Staubli VAL3: Staubli.pjx

--- Staubli.pjx ---
Parameters version=s7.9.1 stackSize=5000 millimeterUnit=true
Program file=decodeVelCfg.pgx
Program file=decodeVelCmd.pgx
Program file=decSetDrvPwrMsg.pgx
Program file=decWriSingIOMsg.pgx
Program file=encodeVelCfgAck.pgx
Program file=encodeVelCmdAck.pgx
Program file=encSetDrvPwrAck.pgx
Program file=encWriSingIOAck.pgx
Program file=init.pgx
Program file=initStaubliMsgs.pgx
Program file=start.pgx
Program file=stop.pgx
Data file=Staubli.dtx
Library alias=SimpleMsg path=Disk://ros_libs/SimpleMessage/SimpleMessage.pjx
Type name=_MotionMode path=./_MotionMode/MotionMode.pjx
Type name=_MsgTypeStaubli path=./_MsgTypeStaubli/MsgTypeStaubli.pjx
Type name=_VelocityType path=./_VelocityType/VelocityType.pjx
Type name=VelocityCmdMsg path=./VelocityCmdMsg/VelocityCmdMsg.pjx
Type name=VelocityCfgMsg path=./VelocityCfgMsg/VelocityCfgMsg.pjx
Type name=SetDrivePwrMsg path=./SetDrivePwrMsg/SetDrivePwrMsg.pjx
Type name=WriteSingIOMsg path=./WriteSingIOMsg/WriteSingIOMsg.pjx

--- Staubli.dtx ---
public SetDrivePwrMsg setDrvPwrAck
  [0]
    bool bDrivePower
    Body body
      [0]
        num nData
    Header header
      [0]
        num nCommType
        num nData[12]
        num nMsgType
        num nReplyCode
    Prefix prefix
      [0]
        num nData[4]
        num nLength
public SetDrivePwrMsg setDrvPwrMsg
  [0]
    bool bDrivePower
    Body body
      [0]
        num nData
    Header header
      [0]
        num nCommType
        num nData[12]
        num nMsgType
        num nReplyCode
    Prefix prefix
      [0]
        num nData[4]
        num nLength
public VelocityCfgMsg velCfgAck
  [0]
    Body body
      [0]
        num nData[68]
    Header header
      [0]
        num nCommType
        num nData[12]
        num nMsgType
        num nReplyCode
    Prefix prefix
      [0]
        num nData[4]
        num nLength = 76
    VelocityCfg velCfg
      [0]
        num nAccel
        num nCmdType
        num nRefFrameVec[6]
        num nRotVel
        num nToolVec[6]
        num nTransVel
public VelocityCfgMsg velCfgMsg
  [0]
    Body body
      [0]
        num nData[68]
    Header header
      [0]
        num nCommType
        num nData[12]
        num nMsgType
        num nReplyCode
    Prefix prefix
      [0]
        num nData[4]
        num nLength
    VelocityCfg velCfg
      [0]
        num nAccel
        num nCmdType
        num nRefFrameVec[6]
        num nRotVel
        num nToolVec[6]
        num nTransVel
public VelocityCmdMsg velCmdAck
  [0]
    Body body
      [0]
        num nData[32]
    Header header
      [0]
        num nCommType
        num nData[12]
        num nMsgType
        num nReplyCode
    Prefix prefix
      [0]
        num nData[4]
        num nLength = 44
    VelocityCmd velCmd
      [0]
        num nCmdType
        num nSeq
        num nVelVec[6]
public VelocityCmdMsg velCmdMsg
  [0]
    Body body
      [0]
        num nData[32]
    Header header
      [0]
        num nCommType
        num nData[12]
        num nMsgType
        num nReplyCode
    Prefix prefix
      [0]
        num nData[4]
        num nLength
    VelocityCmd velCmd
      [0]
        num nCmdType
        num nSeq
        num nVelVec[6]
public WriteSingIOMsg writeSingIOMsg
  [0]
    Body body
      [0]
        num nData[9]
    Header header
      [0]
        num nCommType
        num nData[12]
        num nMsgType
        num nReplyCode
    Prefix prefix
      [0]
        num nData[4]
        num nLength
    WriteSingleIO writeSingleIO
      [0]
        bool bState
        num nModuleId
        num nPin
public WriteSingIOMsg writeSingIOAck
  [0]
    Body body
      [0]
        num nData[9]
    Header header
      [0]
        num nCommType
        num nData[12]
        num nMsgType
        num nReplyCode
    Prefix prefix
      [0]
        num nData[4]
        num nLength
    WriteSingleIO writeSingleIO
      [0]
        bool bState
        num nModuleId
        num nPin
public _MotionMode MotionMode
  [0]
    num INVALID
    num JOINT_TRAJ = 1
    num VELOCITY_CTRL = 4
public _MsgTypeStaubli MsgType
  [0]
    num SET_DRIVE_POWER
    num VELOCITY_CFG = 1640
    num VELOCITY_CMD = 1641
    num READ_IO
    num WRITE_SINGLE_IO
public _VelocityType VelocityType
  [0]
    num INVALID
    num JOINT = 1
    num BASE_FRAME = 2
    num TOOL_FRAME = 3

--- decodeVelCfg.pgx ---
public program decodeVelCfg(bool& x_bFlag (dimensions=1))
  local num l_nIndex
  local num l_nRetVal
begin
  // Copyright (c) 2021, Institute for Factory Automation and Production Systems (FAPS)
  //
  // Licensed under the Apache License, Version 2.0 (the "License");
  // you may not use this file except in compliance with the License.
  // You may obtain a copy of the License at
  //
  //     http://www.apache.org/licenses/LICENSE-2.0
  //
  // Unless required by applicable law or agreed to in writing, software
  // distributed under the License is distributed on an "AS IS" BASIS,
  // WITHOUT WARRANTIES OR CONDITIONS OF ANY KIND, either express or implied.
  // See the License for the specific language governing permissions and
  // limitations under the License.


  // decode velocity configuration message body (data)

  // assume failure to decode
  velCfgAck.header.nReplyCode=SimpleMsg:ReplyCode.FAILURE


  // command type (frame or joint), 4 bytes
  l_nRetVal=fromBinary(velCfgMsg.body.nData,4,"-4l",velCfgMsg.velCfg.nCmdType)
  if (l_nRetVal!=1)
    x_bFlag=false
    return
  endIf

  // reference frame vector [6], 24 bytes
  for l_nIndex=0 to 5 step 1
    l_nRetVal=fromBinary(velCfgMsg.body.nData[(l_nIndex*4)+4],4,"4.0l",velCfgMsg.velCfg.nRefFrameVec[l_nIndex])
    if (l_nRetVal!=1)
      x_bFlag=false
      return
    endIf
  endFor

  // target tool vector [6], 24 bytes
  for l_nIndex=0 to 5 step 1
    l_nRetVal=fromBinary(velCfgMsg.body.nData[(l_nIndex*4)+28],4,"4.0l",velCfgMsg.velCfg.nToolVec[l_nIndex])
    if (l_nRetVal!=1)
      x_bFlag=false
      return
    endIf
  endFor

  // acceleration, 4 bytes
  l_nRetVal=fromBinary(velCfgMsg.body.nData[52],4,"4.0l",velCfgMsg.velCfg.nAccel)
  if (l_nRetVal!=1)
    x_bFlag=false
    return
  endIf

  // velocity, 4 bytes
  l_nRetVal=fromBinary(velCfgMsg.body.nData[56],4,"4.0l",velCfgMsg.velCfg.nVel)
  if (l_nRetVal!=1)
    x_bFlag=false
    return
  endIf

  // translational velocity, 4 bytes
  l_nRetVal=fromBinary(velCfgMsg.body.nData[60],4,"4.0l",velCfgMsg.velCfg.nTransVel)
  if (l_nRetVal!=1)
    x_bFlag=false
    return
  endIf

  // rotational velocity, 4 bytes
  l_nRetVal=fromBinary(velCfgMsg.body.nData[64],4,"4.0l",velCfgMsg.velCfg.nRotVel)
  if (l_nRetVal!=1)
    x_bFlag=false
    return
  endIf


  // decoding successful
  velCfgAck.header.nReplyCode=SimpleMsg:ReplyCode.SUCCESS
  velCfgAck.velCfg.nCmdType=velCfgMsg.velCfg.nCmdType
  x_bFlag=true
end

--- decodeVelCmd.pgx ---
public program decodeVelCmd(bool& x_bFlag (dimensions=1))
  local num l_nIndex
  local num l_nRetVal
begin
  // Copyright (c) 2021, Institute for Factory Automation and Production Systems (FAPS)
  //
  // Licensed under the Apache License, Version 2.0 (the "License");
  // you may not use this file except in compliance with the License.
  // You may obtain a copy of the License at
  //
  //     http://www.apache.org/licenses/LICENSE-2.0
  //
  // Unless required by applicable law or agreed to in writing, software
  // distributed under the License is distributed on an "AS IS" BASIS,
  // WITHOUT WARRANTIES OR CONDITIONS OF ANY KIND, either express or implied.
  // See the License for the specific language governing permissions and
  // limitations under the License.


  // decode velocity command message body (data)

  // assume failure to decode
  velCmdAck.header.nReplyCode=SimpleMsg:ReplyCode.FAILURE


  // sequence, 4 bytes
  l_nRetVal=fromBinary(velCmdMsg.body.nData,4,"-4l",velCmdMsg.velCmd.nSeq)
  if (l_nRetVal!=1)
    x_bFlag=false
    return
  endIf

  // velocity vector [6], 24 bytes
  for l_nIndex=0 to 5 step 1
    l_nRetVal=fromBinary(velCmdMsg.body.nData[(l_nIndex*4)+4],4,"4.0l",velCmdMsg.velCmd.nVelVec[l_nIndex])
    if (l_nRetVal!=1)
      x_bFlag=false
      return
    endIf
  endFor

  // velocity command type (see Staubli:VelocityType "enum"), 4 bytes
  l_nRetVal=fromBinary(velCmdMsg.body.nData[28],4,"4l",velCmdMsg.velCmd.nCmdType)
  if (l_nRetVal!=1)
    x_bFlag=false
    return
  endIf


  // decoding successful
  velCmdAck.header.nReplyCode=SimpleMsg:ReplyCode.SUCCESS
  velCmdAck.velCmd.nSeq=velCmdMsg.velCmd.nSeq
  x_bFlag=true
end

--- decSetDrvPwrMsg.pgx ---
public program decSetDrvPwrMsg(bool& x_bFlag (dimensions=1))
  local num l_nData
  local num l_nIndex
  local num l_nRetVal
begin
  // Copyright (c) 2021, Institute for Factory Automation and Production Systems (FAPS)
  //
  // Licensed under the Apache License, Version 2.0 (the "License");
  // you may not use this file except in compliance with the License.
  // You may obtain a copy of the License at
  //
  //     http://www.apache.org/licenses/LICENSE-2.0
  //
  // Unless required by applicable law or agreed to in writing, software
  // distributed under the License is distributed on an "AS IS" BASIS,
  // WITHOUT WARRANTIES OR CONDITIONS OF ANY KIND, either express or implied.
  // See the License for the specific language governing permissions and
  // limitations under the License.


  // decode set drive power message body (data)

  // assume failure to decode
  setDrvPwrAck.header.nReplyCode=SimpleMsg:ReplyCode.FAILURE

  // fields:
  //  setDrvPwrMsg.bDrivePower


  // drive power, 1 byte
  l_nRetVal=fromBinary(setDrvPwrMsg.body.nData,1,"1",l_nData)

  if (l_nRetVal!=1)
    x_bFlag=false
    return
  endIf

  if (l_nData==1)
    setDrvPwrMsg.bDrivePower=true
  elseIf (l_nData==0)
    setDrvPwrMsg.bDrivePower=false
  else
    // TODO: debug output
    x_bFlag=false
    return
  endIf

  // decoding successful
  setDrvPwrAck.header.nReplyCode=SimpleMsg:ReplyCode.SUCCESS
  x_bFlag=true
end

--- decWriSingIOMsg.pgx ---
public program decWriSingIOMsg(bool& x_bFlag (dimensions=1))
  local num l_nData
  local num l_nIndex
  local num l_nRetVal
begin
  // Copyright (c) 2021, Institute for Factory Automation and Production Systems (FAPS)
  //
  // Licensed under the Apache License, Version 2.0 (the "License");
  // you may not use this file except in compliance with the License.
  // You may obtain a copy of the License at
  //
  //     http://www.apache.org/licenses/LICENSE-2.0
  //
  // Unless required by applicable law or agreed to in writing, software
  // distributed under the License is distributed on an "AS IS" BASIS,
  // WITHOUT WARRANTIES OR CONDITIONS OF ANY KIND, either express or implied.
  // See the License for the specific language governing permissions and
  // limitations under the License.


  // decode write single IO message body (data)

  // assume failure to decode
  writeSingIOMsg.header.nReplyCode=SimpleMsg:ReplyCode.FAILURE

  // fields:
  //  writeSingIOMsg.writeSingleIO.nModuleId
  //  writeSingIOMsg.writeSingleIO.nPin
  //  writeSingIOMsg.writeSingleIO.bState


  // module id, 4 bytes
  l_nRetVal=fromBinary(writeSingIOMsg.body.nData,1,"-4l",writeSingIOMsg.writeSingleIO.nModuleId)

  if (l_nRetVal!=1)
    x_bFlag=false
    return
  endIf

  // pin, 4 bytes
  l_nRetVal=fromBinary(writeSingIOMsg.body.nData[4],1,"-4l",writeSingIOMsg.writeSingleIO.nPin)

  if (l_nRetVal!=1)
    x_bFlag=false
    return
  endIf

  // state, 1 byte
  l_nRetVal=fromBinary(writeSingIOMsg.body.nData[8],1,"1",l_nData)

  if (l_nRetVal!=1)
    x_bFlag=false
    return
  endIf

  // convert decoded data to bool
  if (l_nData==1)
    writeSingIOMsg.writeSingleIO.bState=true
  elseIf (l_nData==0)
    writeSingIOMsg.writeSingleIO.bState=false
  else
    logMsg("[ERROR] WriteSingleIO.bState was decoded to: "+toString("",l_nData))
    x_bFlag=false
    return
  endIf

  // decoding successful
  writeSingIOAck.header.nReplyCode=SimpleMsg:ReplyCode.SUCCESS
  x_bFlag=true
end

--- encodeVelCfgAck.pgx ---
public program encodeVelCfgAck()
begin
  // Copyright (c) 2021, Institute for Factory Automation and Production Systems (FAPS)
  //
  // Licensed under the Apache License, Version 2.0 (the "License");
  // you may not use this file except in compliance with the License.
  // You may obtain a copy of the License at
  //
  //     http://www.apache.org/licenses/LICENSE-2.0
  //
  // Unless required by applicable law or agreed to in writing, software
  // distributed under the License is distributed on an "AS IS" BASIS,
  // WITHOUT WARRANTIES OR CONDITIONS OF ANY KIND, either express or implied.
  // See the License for the specific language governing permissions and
  // limitations under the License.


  // encode 'prefix' and 'header'
  call SimpleMsg:encPrefixHeader(velCfgAck.prefix,velCfgAck.header)

  // encodings of the body field (dummy data) is ignored to save CPU time, since values are all zeros
end

--- encodeVelCmdAck.pgx ---
public program encodeVelCmdAck()
begin
  // Copyright (c) 2021, Institute for Factory Automation and Production Systems (FAPS)
  //
  // Licensed under the Apache License, Version 2.0 (the "License");
  // you may not use this file except in compliance with the License.
  // You may obtain a copy of the License at
  //
  //     http://www.apache.org/licenses/LICENSE-2.0
  //
  // Unless required by applicable law or agreed to in writing, software
  // distributed under the License is distributed on an "AS IS" BASIS,
  // WITHOUT WARRANTIES OR CONDITIONS OF ANY KIND, either express or implied.
  // See the License for the specific language governing permissions and
  // limitations under the License.


  // encode 'prefix' and 'header'
  call SimpleMsg:encPrefixHeader(velCmdAck.prefix,velCmdAck.header)

  // encode 'body' (data)
  toBinary(velCmdAck.velCmd.nSeq,1,"4l",velCmdAck.body.nData)

  // encodings of the remaining elements (dummy data) is ignored to save CPU time, since values are all zeros
end

--- encSetDrvPwrAck.pgx ---
public program encSetDrvPwrAck()
begin
  // Copyright (c) 2021, Institute for Factory Automation and Production Systems (FAPS)
  //
  // Licensed under the Apache License, Version 2.0 (the "License");
  // you may not use this file except in compliance with the License.
  // You may obtain a copy of the License at
  //
  //     http://www.apache.org/licenses/LICENSE-2.0
  //
  // Unless required by applicable law or agreed to in writing, software
  // distributed under the License is distributed on an "AS IS" BASIS,
  // WITHOUT WARRANTIES OR CONDITIONS OF ANY KIND, either express or implied.
  // See the License for the specific language governing permissions and
  // limitations under the License.


  // encode 'prefix' and 'header'
  call SimpleMsg:encPrefixHeader(setDrvPwrAck.prefix,setDrvPwrAck.header)

  // encodings of the body field (dummy data) is ignored to save CPU time, since values are all zeros
end

--- encWriSingIOAck.pgx ---
public program encWriSingIOAck()
begin
  // Copyright (c) 2021, Institute for Factory Automation and Production Systems (FAPS)
  //
  // Licensed under the Apache License, Version 2.0 (the "License");
  // you may not use this file except in compliance with the License.
  // You may obtain a copy of the License at
  //
  //     http://www.apache.org/licenses/LICENSE-2.0
  //
  // Unless required by applicable law or agreed to in writing, software
  // distributed under the License is distributed on an "AS IS" BASIS,
  // WITHOUT WARRANTIES OR CONDITIONS OF ANY KIND, either express or implied.
  // See the License for the specific language governing permissions and
  // limitations under the License.


  // encode 'prefix' and 'header'
  call SimpleMsg:encPrefixHeader(writeSingIOAck.prefix,writeSingIOAck.header)

  // encodings of the body field (dummy data) is ignored to save CPU time, since values are all zeros
end

--- init.pgx ---
public program init()
begin
  // Copyright (c) 2021, Institute for Factory Automation and Production Systems (FAPS)
  //
  // Licensed under the Apache License, Version 2.0 (the "License");
  // you may not use this file except in compliance with the License.
  // You may obtain a copy of the License at
  //
  //     http://www.apache.org/licenses/LICENSE-2.0
  //
  // Unless required by applicable law or agreed to in writing, software
  // distributed under the License is distributed on an "AS IS" BASIS,
  // WITHOUT WARRANTIES OR CONDITIONS OF ANY KIND, either express or implied.
  // See the License for the specific language governing permissions and
  // limitations under the License.


  // initialize Staubli specific message IDs for the simple message protocol
  MsgType.SET_DRIVE_POWER=1610
  MsgType.READ_IO=1620
  MsgType.WRITE_SINGLE_IO=1621
  MsgType.VELOCITY_CFG=1640
  MsgType.VELOCITY_CMD=1641

  // initialize "enum" values for different motion modes
  MotionMode.INVALID=0
  MotionMode.JOINT_TRAJ=1
  MotionMode.VELOCITY_CTRL=2

  // initialize "enum" values for the three different types of velocity init functions $velJoint, $velFrame, $velTool
  VelocityType.INVALID=0
  VelocityType.JOINT=1
  VelocityType.BASE_FRAME=2
  VelocityType.TOOL_FRAME=3

  // initialize Staubli specific messages (MUST be called last because of the dependency on the values above)
  call initStaubliMsgs()
end

--- initStaubliMsgs.pgx ---
program initStaubliMsgs()
begin
  // Copyright (c) 2021, Institute for Factory Automation and Production Systems (FAPS)
  //
  // Licensed under the Apache License, Version 2.0 (the "License");
  // you may not use this file except in compliance with the License.
  // You may obtain a copy of the License at
  //
  //     http://www.apache.org/licenses/LICENSE-2.0
  //
  // Unless required by applicable law or agreed to in writing, software
  // distributed under the License is distributed on an "AS IS" BASIS,
  // WITHOUT WARRANTIES OR CONDITIONS OF ANY KIND, either express or implied.
  // See the License for the specific language governing permissions and
  // limitations under the License.


  // initialize Staubli specific messages (outgoing)


  // Set drive power message:
  // prefix length = 12 + 1 = 13
  setDrvPwrAck.prefix.nLength=13
  setDrvPwrAck.header.nMsgType=MsgType.SET_DRIVE_POWER
  setDrvPwrAck.header.nCommType=SimpleMsg:CommType.SERVICE_REPLY
  setDrvPwrAck.header.nReplyCode=SimpleMsg:ReplyCode.INVALID
  // body (data) assumed to be initialized to zero


  // Write single IO message:
  // prefix length = 12 + 9 = 21
  writeSingIOAck.prefix.nLength=21
  writeSingIOAck.header.nMsgType=MsgType.WRITE_SINGLE_IO
  writeSingIOAck.header.nCommType=SimpleMsg:CommType.SERVICE_REPLY
  writeSingIOAck.header.nReplyCode=SimpleMsg:ReplyCode.INVALID
  // body (data) assumed to be initialized to zero


  // Velocity mode configuration message:
  // prefix length = 12 + 68 = 80
  velCfgAck.prefix.nLength=80
  velCfgAck.header.nMsgType=MsgType.VELOCITY_CFG
  velCfgAck.header.nCommType=SimpleMsg:CommType.SERVICE_REPLY
  velCfgAck.header.nReplyCode=SimpleMsg:ReplyCode.INVALID
  // body (data) assumed to be initialized to zero


  // Velocity command message:
  // prefix length = 12 + 32 = 44
  velCmdAck.prefix.nLength=44
  velCmdAck.header.nMsgType=MsgType.VELOCITY_CMD
  velCmdAck.header.nCommType=SimpleMsg:CommType.SERVICE_REPLY
  velCmdAck.header.nReplyCode=SimpleMsg:ReplyCode.INVALID
  // body (data) assumed to be initialized to zero
end
